// TIA Portal V20 export
VAR_GLOBAL   // PLC tag table "PFE"
END_VAR
